GLOBALCONSTANTS DefaultPool_Tester (* Global constants *)
  PACKAGE Uebungen::const::UT::Tester;
  VAR_GLOBAL CONSTANT
    ISO_DESIGNATOR_WIDTH : UINT := 80;
    ISO_DESIGNATOR_HEIGHT : UINT := 80;
    ISO_MASK_SIZE : UINT := 480;
    ISO_VERSION_LABEL : STRING;
    MASK_WIDTH : UINT := 480;
    MASK_HEIGHT : UINT := 480;
    WorkingSet : UINT := 0;
    DataMask_M1 : UINT := 1000;
    Container_Q : UINT := 3000;
    Container_I : UINT := 3001;
    Button_Q01 : UINT := 6001;
    Button_Q02 : UINT := 6002;
    Button_Q03 : UINT := 6003;
    Button_Q04 : UINT := 6004;
    Button_Q05 : UINT := 6005;
    Button_Q06 : UINT := 6006;
    Button_Q07 : UINT := 6007;
    Button_Q08 : UINT := 6008;
    Button_Q09 : UINT := 6009;
    Button_Q10 : UINT := 6010;
    Button_Q11 : UINT := 6011;
    Button_Q12 : UINT := 6012;
    Button_I01 : UINT := 6101;
    Button_I02 : UINT := 6102;
    Button_I03 : UINT := 6103;
    Button_I04 : UINT := 6104;
    Button_I05 : UINT := 6105;
    Button_I06 : UINT := 6106;
    Button_I07 : UINT := 6107;
    Button_I08 : UINT := 6108;
    OutputString_WorkingSet_0 : UINT := 11000;
    OutputNumber_12000 : UINT := 12000;
    OutputNumber_12001 : UINT := 12001;
    OutputNumber_12002 : UINT := 12002;
    OutputNumber_12003 : UINT := 12003;
    OutputNumber_12004 : UINT := 12004;
    OutputNumber_12005 : UINT := 12005;
    OutputNumber_12006 : UINT := 12006;
    OutputNumber_12007 : UINT := 12007;
    OutputNumber_12008 : UINT := 12008;
    OutputNumber_12009 : UINT := 12009;
    OutputNumber_12010 : UINT := 12010;
    OutputNumber_12011 : UINT := 12011;
    OutputNumber_12012 : UINT := 12012;
    OutputNumber_12013 : UINT := 12013;
    OutputNumber_12014 : UINT := 12014;
    OutputNumber_12015 : UINT := 12015;
    OutputNumber_12016 : UINT := 12016;
    OutputNumber_12017 : UINT := 12017;
    OutputNumber_12018 : UINT := 12018;
    OutputNumber_12019 : UINT := 12019;
    Logos_icon : UINT := 20500;
    FontAttributes_6x8 : UINT := 23000;
    FontAttributes_24x32 : UINT := 23001;
    AuxFunction2_X1 : UINT := 31000;
  END_VAR
END_GLOBALCONSTANTS
